(* Logix 5000 project; controller Receptivo vendor 1 type 14 code 106 rev 30.11; software revision 30.00; part 4 of 10 *)
(* tags used below, declared in another part *)
   Bit_Medianoche : BOOL;
   bit_ptobar : BOOL;
   Calendario : Hora_y_Fecha;
   Cola_Densidad_Bidon_Ayer : REAL[50];
   Cola_Densidad_Bidon_Fecha_Ayer : Hora_y_Fecha[50];
   Cola_Densidad_Bidones : REAL[50];
   Cola_Densidad_Bidones_Fecha : Hora_y_Fecha[50];
   Cola_Densidad_Elmar : REAL[50];
   Cola_Densidad_Elmar_Ayer : REAL[50];
   Cola_Densidad_Elmar_Fecha : Hora_y_Fecha[50];
   Cola_Densidad_Elmar_Fecha_Ayer : Hora_y_Fecha[50];
   Cola_Densidad_Fogg1 : REAL[50];
   Cola_Densidad_Fogg1_Ayer : REAL[50];
   Cola_Densidad_fogg1_Fecha : Hora_y_Fecha[50];
   Cola_Densidad_fogg1_Fecha_Ayer : Hora_y_Fecha[50];
   Cola_Densidad_Fogg2 : REAL[50];
   Cola_Densidad_Fogg2_Ayer : REAL[50];
   Cola_Densidad_fogg2_Fecha : Hora_y_Fecha[50];
   Cola_Densidad_fogg2_Fecha_Ayer : Hora_y_Fecha[50];
   Cola_Densidad_Karat : REAL[50];
   Cola_Densidad_Karat_Ayer : REAL[50];
   Cola_Densidad_Karat_Fecha : Hora_y_Fecha[50];
   Cola_Densidad_Karat_Fecha_Ayer : Hora_y_Fecha[50];
   Cola_Peso_Bidones : REAL[50];
   Cola_Peso_Caja_Bidon_Ayer : REAL[50];
   Cola_Peso_Caja_Elmar : REAL[50];
   Cola_Peso_Caja_Elmar_Ayer : REAL[50];
   Cola_Peso_Caja_Fogg1 : REAL[50];
   Cola_Peso_Caja_Fogg1_Ayer : REAL[50];
   Cola_Peso_Caja_Fogg2 : REAL[50];
   Cola_Peso_Caja_Fogg2_Ayer : REAL[50];
   Cola_Peso_Caja_Karat : REAL[50];
   Cola_Peso_Caja_Karat_Ayer : REAL[50];
   Cola_QAD_Densidad_Bidon_Ayer : STRING[50];
   Cola_QAD_Densidad_Bidones : STRING[50];
   Cola_QAD_Densidad_Elmar : STRING[50];
   Cola_QAD_Densidad_Elmar_Ayer : STRING[50];
   Cola_QAD_Densidad_Fogg1 : STRING[50];
   Cola_QAD_Densidad_Fogg1_Ayer : STRING[50];
   Cola_QAD_Densidad_Fogg2 : STRING[50];
   Cola_QAD_Densidad_Fogg2_Ayer : STRING[50];
   Cola_QAD_Densidad_Karat : STRING[50];
   Cola_QAD_Densidad_Karat_Ayer : STRING[50];
   Control_Densidad_Bidones : CONTROL;
   Control_Densidad_Elmar : CONTROL;
   Control_Densidad_Fogg1 : CONTROL;
   Control_Densidad_Fogg2 : CONTROL;
   Control_Densidad_Karat : CONTROL;
   Densidad_Bidon_1 : REAL;
   Densidad_Bidones : REAL;
   Densidad_Elmar : REAL;
   Densidad_Elmar_1 : REAL;
   Densidad_Elmar_OK : BOOL;
   Densidad_Fogg1 : REAL;
   Densidad_Fogg1_1 : REAL;
   Densidad_Fogg1_OK : BOOL;
   Densidad_Fogg2 : REAL;
   Densidad_Fogg2_1 : REAL;
   Densidad_Fogg2_OK : BOOL;
   Densidad_Karat : REAL;
   Densidad_Karat_1 : REAL;
   Densidad_Karat_OK : BOOL;
   Hora_Ingreso_Datos_Elmar : Hora_y_Fecha;
   Index_Bidones_Videojet : DINT;
   Index_Elmar_Videojet : DINT;
   Index_Fogg1_Videojet : DINT;
   Index_Fogg2_Videojet : DINT;
   Index_Karat_Videojet : DINT;
   Index_Karat_Videojet_Antiguo : DINT;
   Lote : DINT;
   Nuevo_Lote_Fogg1 : BOOL;
   ons_datos_mal_Bidones : BOOL;
   ons_datos_mal_elmar : BOOL;
   ons_datos_mal_Fogg1 : BOOL;
   ons_datos_mal_Fogg2 : BOOL;
   Ons_Datos_Mal_Karat : BOOL;
   ons_densidad_Fogg_1 : BOOL;
   Ons_Nuevo_Karat_Videojet : BOOL;
   Pesaje_Elmar_OK : BOOL;
   Pesaje_Fogg1_OK : BOOL;
   Pesaje_Fogg2_OK : BOOL;
   Pesaje_Karat_OK : BOOL;
   Peso_Bidones : REAL;
   Peso_Bidones_1 : REAL;
   Peso_Caja_Elmar : REAL;
   Peso_Caja_Elmar_1 : REAL;
   Peso_Caja_Fogg1 : REAL;
   Peso_Caja_Fogg1_1 : REAL;
   Peso_Caja_Fogg2 : REAL;
   Peso_Caja_Fogg2_1 : REAL;
   Peso_Caja_Karat : REAL;
   Peso_Caja_Karat_1 : REAL;
   Producido_Bidones_Ahora : UDT_Maestro;
   Producido_Elmar_Ahora : UDT_Maestro;
   Producido_Fogg1_Ahora : UDT_Maestro;
   Producido_Fogg2_Ahora : UDT_Maestro;
   Producido_Karat_Ahora : UDT_Maestro;
   Productos : UDT_Maestro[300];
   PV_Datos_Mal_Bidones : BOOL;
   PV_Datos_Mal_Elmar : BOOL;
   PV_Datos_Mal_Fogg1 : BOOL;
   PV_Datos_Mal_Fogg2 : BOOL;
   PV_Datos_Mal_Karat : BOOL;
   PV_Datos_Malos_Elmar : BOOL;
   PV_Datos_Malos_Fogg2 : BOOL;
   PV_Datos_Malos_Karat : BOOL;
   PV_Datos_Pesaje_Bidones : BOOL;
   PV_Datos_Pesaje_Elmar : BOOL;
   PV_Datos_Pesaje_Fogg1 : BOOL;
   PV_Datos_Pesaje_Fogg2 : BOOL;
   PV_Datos_Pesaje_Karat : BOOL;
   Slash : STRING;
   Timer_Datos_Bidones : TIMER;
   U_Fecha_Bidones : Hora_y_Fecha;
   U_Fecha_Elmar : Hora_y_Fecha;
   U_Fecha_Fogg1 : Hora_y_Fecha;
   U_Fecha_Fogg2 : Hora_y_Fecha;
   U_Fecha_Karat : Hora_y_Fecha;
   Un_Espacio : STRING;

PROGRAM Calculo_Produccion   (* main routine Principal_Calculo *)
VAR
   Entro_Datos_Pesaje_Bidones : BOOL;
   Entro_Datos_Pesaje_Elmar : BOOL;
   Entro_Datos_Pesaje_Fogg1 : BOOL;
   Entro_Datos_Pesaje_Fogg2 : BOOL;
   Entro_Datos_Pesaje_Karat : BOOL;
   Fecha_Cero : Hora_y_Fecha;
   Index_Bidones_Videojet_Antiguo : DINT;
   Index_Elmar_Videojet_Antiguo : DINT := 112;
   Index_Fogg1_Videojet_Antiguo : DINT := 203;
   Index_Fogg2_Videojet_Antiguo : DINT := 23;
   Nuevo_Lote_Bidones : BOOL;
   Nuevo_Lote_Elmar : BOOL;
   Nuevo_Lote_Fogg2 : BOOL;
   Nuevo_Lote_Karat : BOOL;
   ons_datos_elmar_malos : BOOL;
   ons_datos_fogg1_malos : BOOL;
   ons_datos_fogg2_malos : BOOL;
   Ons_Datos_Malos_Karat : BOOL;
   ons_densidad_bidones : BOOL;
   ons_densidad_elmar_1 : BOOL;
   ons_densidad_Fogg_2 : BOOL;
   Ons_Densidad_Karat : BOOL;
   ons_medianoche_Bidones : BOOL;
   ons_medianoche_Elmar : BOOL;
   ons_medianoche_Fogg1 : BOOL;
   ons_medianoche_Fogg2 : BOOL;
   Ons_Medianoche_Karat : BOOL;
   ons_nuevo_bidones_videojet : BOOL;
   ons_nuevo_elmar_videojet : BOOL;
   ons_nuevo_fogg1_videojet : BOOL;
   ons_nuevo_fogg2_videojet : BOOL;
   ons_peso_caja_elmar_1 : BOOL;
   Peso_Caja_Elmar_Entro : BOOL;
   PV_Datos_Malos_Fogg1 : BOOL;
   Salida_cola_densidad_elmar : REAL;
   Salida_peso_caja_elmar : REAL;
   Timer_Datos_1 : TIMER := (PRE := 600000);
   Timer_Datos_Fogg1 : TIMER := (PRE := 600000);
   Timer_Datos_Fogg2 : TIMER := (PRE := 600000);
   Timer_Datos_Karat : TIMER := (PRE := 600000);
END_VAR

ROUTINE Calculo_Pesaje_Bidones   (* ladder *)
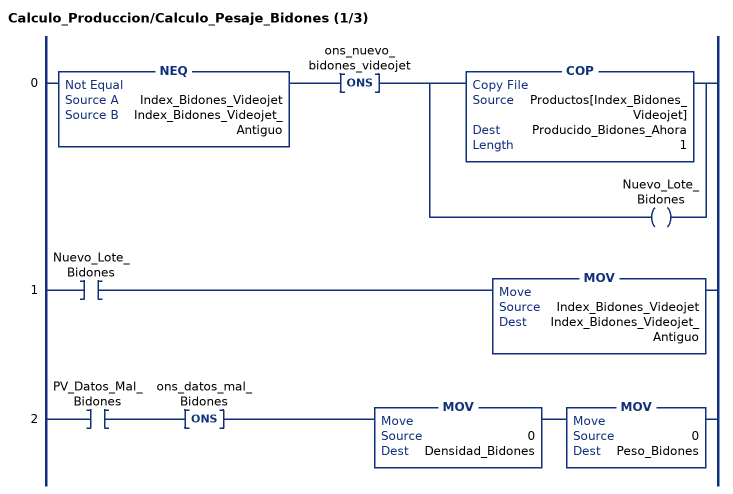
   0: NEQ(Index_Bidones_Videojet,Index_Bidones_Videojet_Antiguo)ONS(ons_nuevo_bidones_videojet)[COP(Productos[Index_Bidones_Videojet],Producido_Bidones_Ahora,1) ,OTE(Nuevo_Lote_Bidones) ];
   1: XIC(Nuevo_Lote_Bidones)MOV(Index_Bidones_Videojet,Index_Bidones_Videojet_Antiguo);
   2: XIC(PV_Datos_Mal_Bidones)ONS(ons_datos_mal_Bidones)MOV(0,Densidad_Bidones)MOV(0,Peso_Bidones);
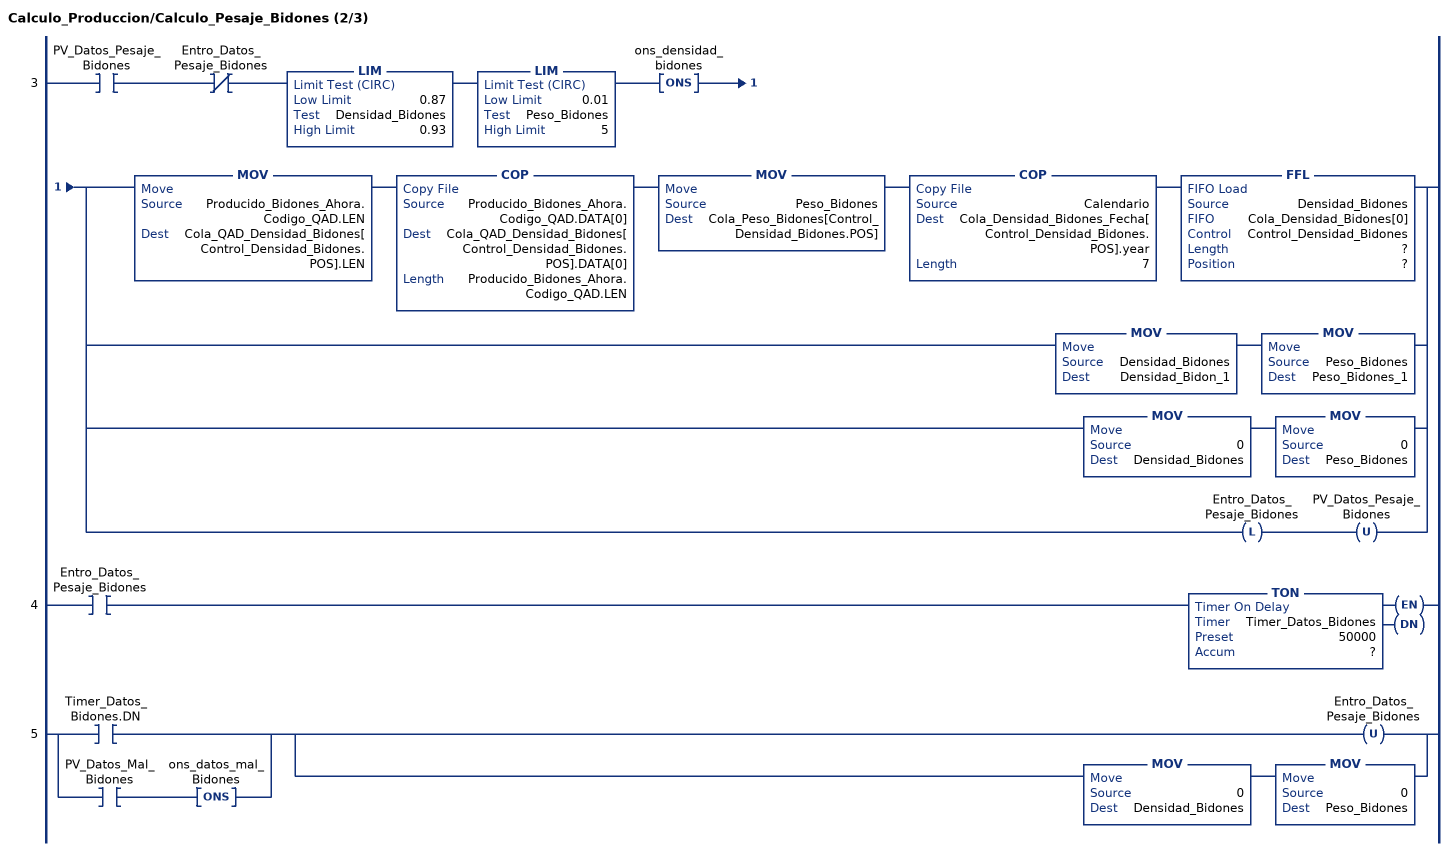
   3: XIC(PV_Datos_Pesaje_Bidones)XIO(Entro_Datos_Pesaje_Bidones)LIM(0.87,Densidad_Bidones,0.93)LIM(0.01,Peso_Bidones,5)ONS(ons_densidad_bidones)[MOV(Producido_Bidones_Ahora.Codigo_QAD.LEN,Cola_QAD_Densidad_Bidones[Control_Densidad_Bidones.POS].LEN) COP(Producido_Bidones_Ahora.Codigo_QAD.DATA[0],Cola_QAD_Densidad_Bidones[Control_Densidad_Bidones.POS].DATA[0],Producido_Bidones_Ahora.Codigo_QAD.LEN) MOV(Peso_Bidones,Cola_Peso_Bidones[Control_Densidad_Bidones.POS]) COP(Calendario,Cola_Densidad_Bidones_Fecha[Control_Densidad_Bidones.POS].year,7) FFL(Densidad_Bidones,Cola_Densidad_Bidones[0],Control_Densidad_Bidones,?,?) ,MOV(Densidad_Bidones,Densidad_Bidon_1) MOV(Peso_Bidones,Peso_Bidones_1) ,MOV(0,Densidad_Bidones) MOV(0,Peso_Bidones) ,OTL(Entro_Datos_Pesaje_Bidones) OTU(PV_Datos_Pesaje_Bidones) ];
   4: XIC(Entro_Datos_Pesaje_Bidones)TON(Timer_Datos_Bidones,?,?);
   5: [XIC(Timer_Datos_Bidones.DN) ,XIC(PV_Datos_Mal_Bidones) ONS(ons_datos_mal_Bidones) ][OTU(Entro_Datos_Pesaje_Bidones) ,MOV(0,Densidad_Bidones) MOV(0,Peso_Bidones) ];
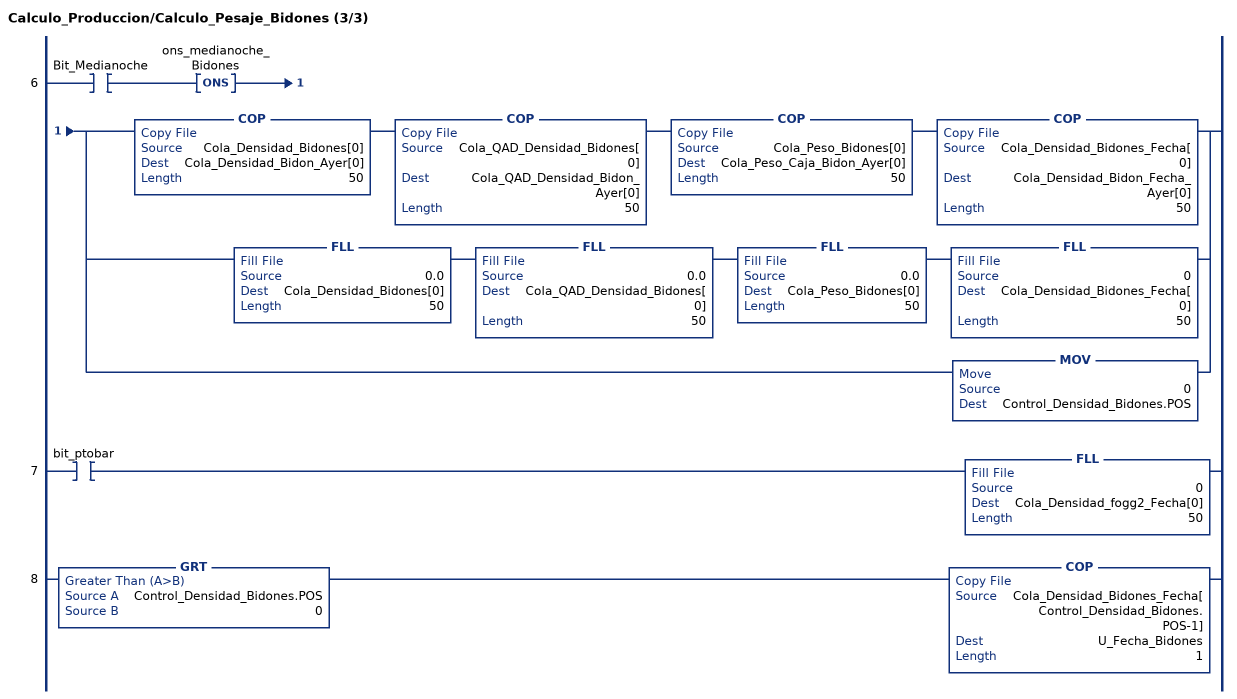
   6: XIC(Bit_Medianoche)ONS(ons_medianoche_Bidones)[COP(Cola_Densidad_Bidones[0],Cola_Densidad_Bidon_Ayer[0],50) COP(Cola_QAD_Densidad_Bidones[0],Cola_QAD_Densidad_Bidon_Ayer[0],50) COP(Cola_Peso_Bidones[0],Cola_Peso_Caja_Bidon_Ayer[0],50) COP(Cola_Densidad_Bidones_Fecha[0],Cola_Densidad_Bidon_Fecha_Ayer[0],50) ,FLL(0.0,Cola_Densidad_Bidones[0],50) FLL(0.0,Cola_QAD_Densidad_Bidones[0],50) FLL(0.0,Cola_Peso_Bidones[0],50) FLL(0,Cola_Densidad_Bidones_Fecha[0],50) ,MOV(0,Control_Densidad_Bidones.POS) ];
   7: XIC(bit_ptobar)FLL(0,Cola_Densidad_fogg2_Fecha[0],50);
   8: GRT(Control_Densidad_Bidones.POS,0)COP(Cola_Densidad_Bidones_Fecha[Control_Densidad_Bidones.POS-1],U_Fecha_Bidones,1);
END_ROUTINE

ROUTINE Calculo_Pesaje_Elmar   (* ladder *)
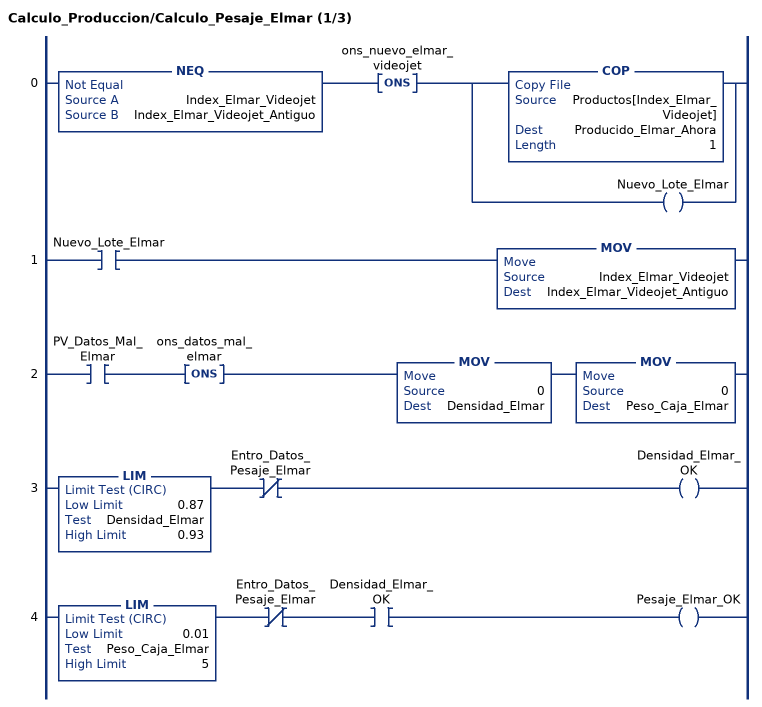
   0: NEQ(Index_Elmar_Videojet,Index_Elmar_Videojet_Antiguo)ONS(ons_nuevo_elmar_videojet)[COP(Productos[Index_Elmar_Videojet],Producido_Elmar_Ahora,1) ,OTE(Nuevo_Lote_Elmar) ];
   1: XIC(Nuevo_Lote_Elmar)MOV(Index_Elmar_Videojet,Index_Elmar_Videojet_Antiguo);
   2: XIC(PV_Datos_Mal_Elmar)ONS(ons_datos_mal_elmar)MOV(0,Densidad_Elmar)MOV(0,Peso_Caja_Elmar);
   3: LIM(0.87,Densidad_Elmar,0.93)XIO(Entro_Datos_Pesaje_Elmar)OTE(Densidad_Elmar_OK);
   4: LIM(0.01,Peso_Caja_Elmar,5)XIO(Entro_Datos_Pesaje_Elmar)XIC(Densidad_Elmar_OK)OTE(Pesaje_Elmar_OK);
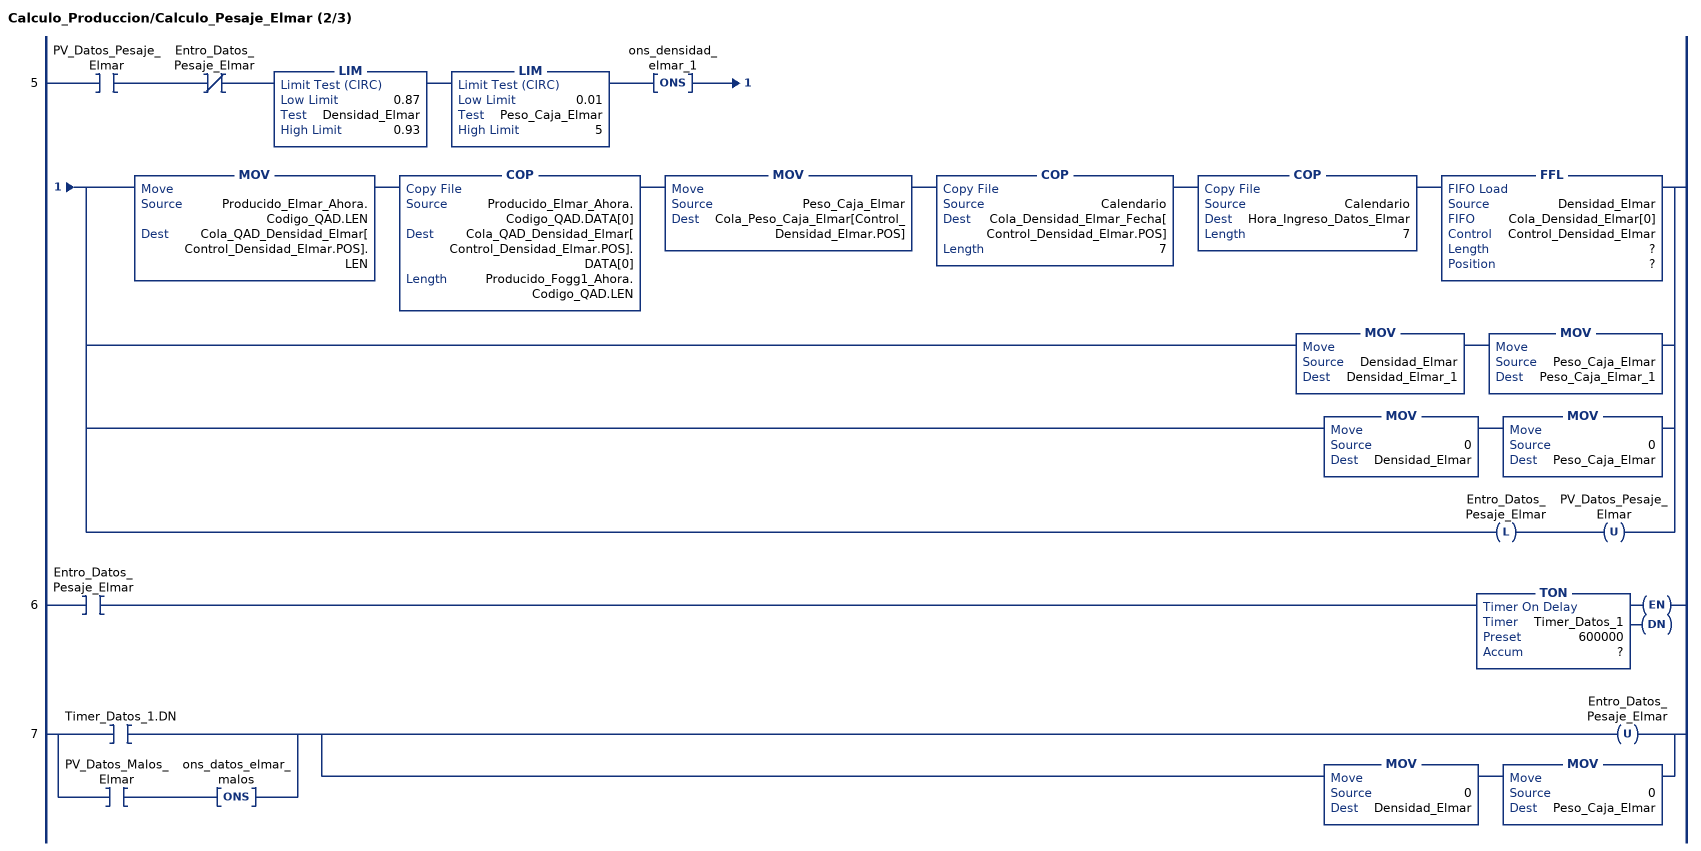
   5: XIC(PV_Datos_Pesaje_Elmar)XIO(Entro_Datos_Pesaje_Elmar)LIM(0.87,Densidad_Elmar,0.93)LIM(0.01,Peso_Caja_Elmar,5)ONS(ons_densidad_elmar_1)[MOV(Producido_Elmar_Ahora.Codigo_QAD.LEN,Cola_QAD_Densidad_Elmar[Control_Densidad_Elmar.POS].LEN) COP(Producido_Elmar_Ahora.Codigo_QAD.DATA[0],Cola_QAD_Densidad_Elmar[Control_Densidad_Elmar.POS].DATA[0],Producido_Fogg1_Ahora.Codigo_QAD.LEN) MOV(Peso_Caja_Elmar,Cola_Peso_Caja_Elmar[Control_Densidad_Elmar.POS]) COP(Calendario,Cola_Densidad_Elmar_Fecha[Control_Densidad_Elmar.POS],7) COP(Calendario,Hora_Ingreso_Datos_Elmar,7) FFL(Densidad_Elmar,Cola_Densidad_Elmar[0],Control_Densidad_Elmar,?,?) ,MOV(Densidad_Elmar,Densidad_Elmar_1) MOV(Peso_Caja_Elmar,Peso_Caja_Elmar_1) ,MOV(0,Densidad_Elmar) MOV(0,Peso_Caja_Elmar) ,OTL(Entro_Datos_Pesaje_Elmar) OTU(PV_Datos_Pesaje_Elmar) ];
   6: XIC(Entro_Datos_Pesaje_Elmar)TON(Timer_Datos_1,?,?);
   7: [XIC(Timer_Datos_1.DN) ,XIC(PV_Datos_Malos_Elmar) ONS(ons_datos_elmar_malos) ][OTU(Entro_Datos_Pesaje_Elmar) ,MOV(0,Densidad_Elmar) MOV(0,Peso_Caja_Elmar) ];
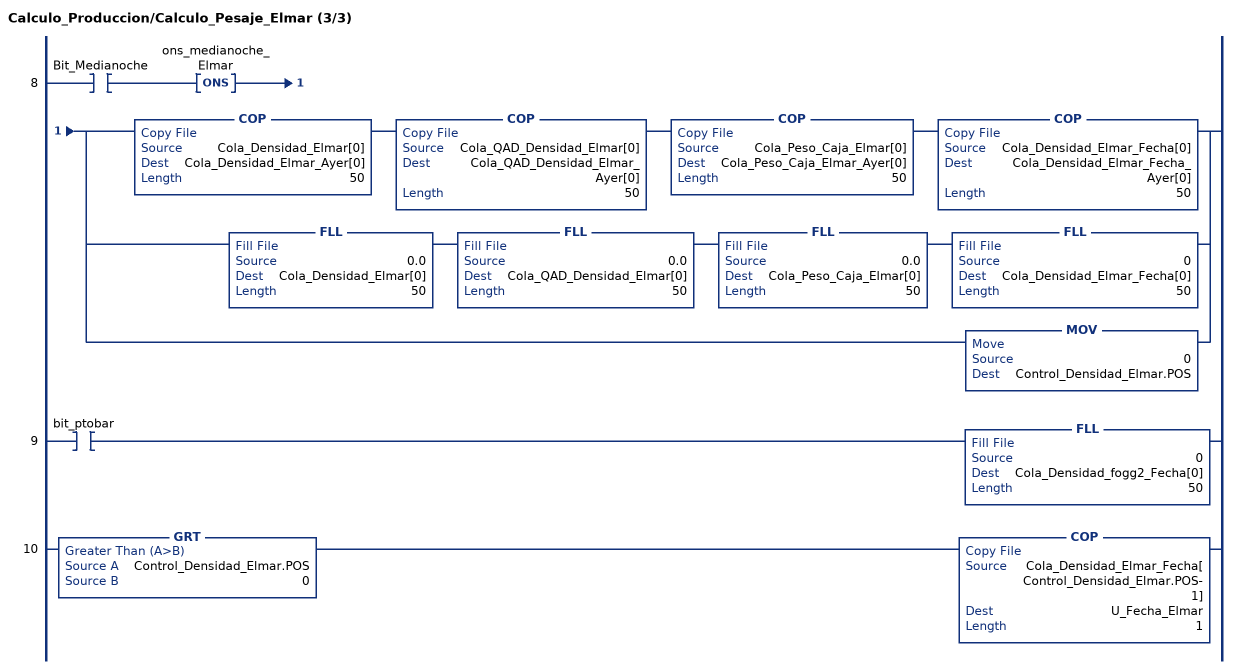
   8: XIC(Bit_Medianoche)ONS(ons_medianoche_Elmar)[COP(Cola_Densidad_Elmar[0],Cola_Densidad_Elmar_Ayer[0],50) COP(Cola_QAD_Densidad_Elmar[0],Cola_QAD_Densidad_Elmar_Ayer[0],50) COP(Cola_Peso_Caja_Elmar[0],Cola_Peso_Caja_Elmar_Ayer[0],50) COP(Cola_Densidad_Elmar_Fecha[0],Cola_Densidad_Elmar_Fecha_Ayer[0],50) ,FLL(0.0,Cola_Densidad_Elmar[0],50) FLL(0.0,Cola_QAD_Densidad_Elmar[0],50) FLL(0.0,Cola_Peso_Caja_Elmar[0],50) FLL(0,Cola_Densidad_Elmar_Fecha[0],50) ,MOV(0,Control_Densidad_Elmar.POS) ];
   9: XIC(bit_ptobar)FLL(0,Cola_Densidad_fogg2_Fecha[0],50);
   10: GRT(Control_Densidad_Elmar.POS,0)COP(Cola_Densidad_Elmar_Fecha[Control_Densidad_Elmar.POS-1],U_Fecha_Elmar,1);
END_ROUTINE

ROUTINE Calculo_Pesaje_Fogg1   (* ladder *)
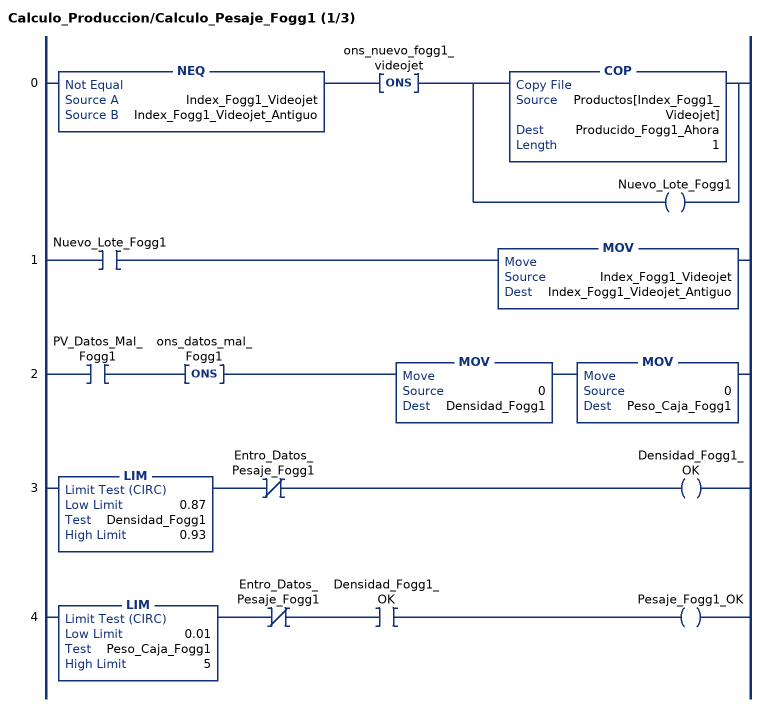
   0: NEQ(Index_Fogg1_Videojet,Index_Fogg1_Videojet_Antiguo)ONS(ons_nuevo_fogg1_videojet)[COP(Productos[Index_Fogg1_Videojet],Producido_Fogg1_Ahora,1) ,OTE(Nuevo_Lote_Fogg1) ];
   1: XIC(Nuevo_Lote_Fogg1)MOV(Index_Fogg1_Videojet,Index_Fogg1_Videojet_Antiguo);
   2: XIC(PV_Datos_Mal_Fogg1)ONS(ons_datos_mal_Fogg1)MOV(0,Densidad_Fogg1)MOV(0,Peso_Caja_Fogg1);
   3: LIM(0.87,Densidad_Fogg1,0.93)XIO(Entro_Datos_Pesaje_Fogg1)OTE(Densidad_Fogg1_OK);
   4: LIM(0.01,Peso_Caja_Fogg1,5)XIO(Entro_Datos_Pesaje_Fogg1)XIC(Densidad_Fogg1_OK)OTE(Pesaje_Fogg1_OK);
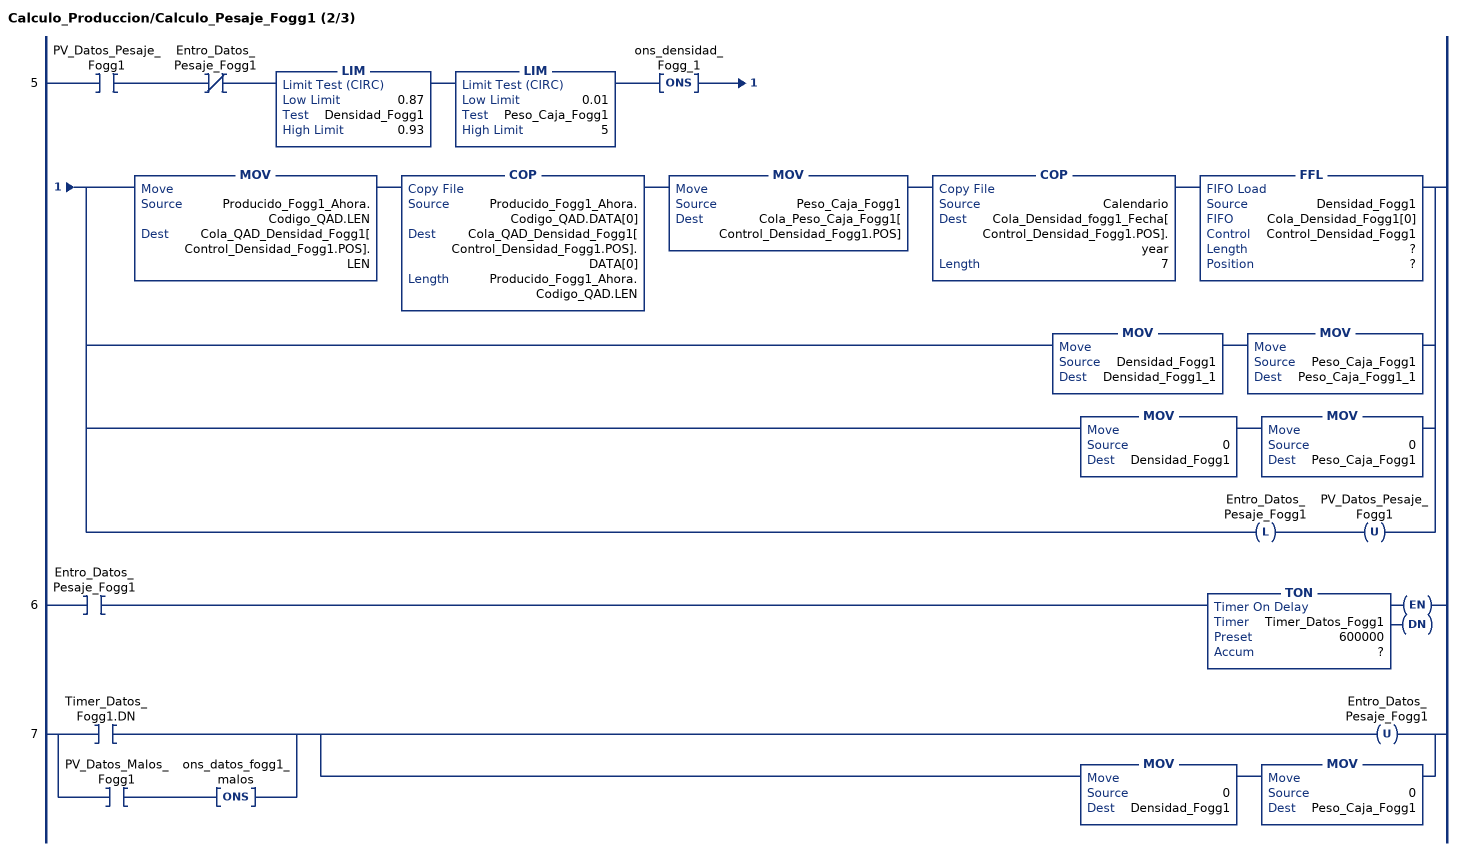
   5: XIC(PV_Datos_Pesaje_Fogg1)XIO(Entro_Datos_Pesaje_Fogg1)LIM(0.87,Densidad_Fogg1,0.93)LIM(0.01,Peso_Caja_Fogg1,5)ONS(ons_densidad_Fogg_1)[MOV(Producido_Fogg1_Ahora.Codigo_QAD.LEN,Cola_QAD_Densidad_Fogg1[Control_Densidad_Fogg1.POS].LEN) COP(Producido_Fogg1_Ahora.Codigo_QAD.DATA[0],Cola_QAD_Densidad_Fogg1[Control_Densidad_Fogg1.POS].DATA[0],Producido_Fogg1_Ahora.Codigo_QAD.LEN) MOV(Peso_Caja_Fogg1,Cola_Peso_Caja_Fogg1[Control_Densidad_Fogg1.POS]) COP(Calendario,Cola_Densidad_fogg1_Fecha[Control_Densidad_Fogg1.POS].year,7) FFL(Densidad_Fogg1,Cola_Densidad_Fogg1[0],Control_Densidad_Fogg1,?,?) ,MOV(Densidad_Fogg1,Densidad_Fogg1_1) MOV(Peso_Caja_Fogg1,Peso_Caja_Fogg1_1) ,MOV(0,Densidad_Fogg1) MOV(0,Peso_Caja_Fogg1) ,OTL(Entro_Datos_Pesaje_Fogg1) OTU(PV_Datos_Pesaje_Fogg1) ];
   6: XIC(Entro_Datos_Pesaje_Fogg1)TON(Timer_Datos_Fogg1,?,?);
   7: [XIC(Timer_Datos_Fogg1.DN) ,XIC(PV_Datos_Malos_Fogg1) ONS(ons_datos_fogg1_malos) ][OTU(Entro_Datos_Pesaje_Fogg1) ,MOV(0,Densidad_Fogg1) MOV(0,Peso_Caja_Fogg1) ];
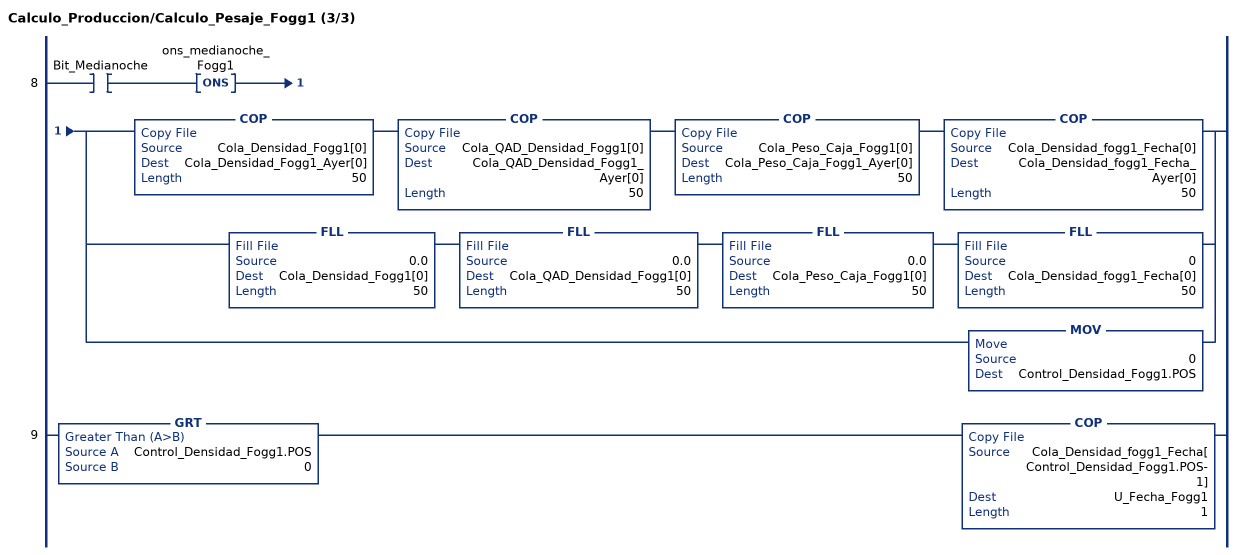
   8: XIC(Bit_Medianoche)ONS(ons_medianoche_Fogg1)[COP(Cola_Densidad_Fogg1[0],Cola_Densidad_Fogg1_Ayer[0],50) COP(Cola_QAD_Densidad_Fogg1[0],Cola_QAD_Densidad_Fogg1_Ayer[0],50) COP(Cola_Peso_Caja_Fogg1[0],Cola_Peso_Caja_Fogg1_Ayer[0],50) COP(Cola_Densidad_fogg1_Fecha[0],Cola_Densidad_fogg1_Fecha_Ayer[0],50) ,FLL(0.0,Cola_Densidad_Fogg1[0],50) FLL(0.0,Cola_QAD_Densidad_Fogg1[0],50) FLL(0.0,Cola_Peso_Caja_Fogg1[0],50) FLL(0,Cola_Densidad_fogg1_Fecha[0],50) ,MOV(0,Control_Densidad_Fogg1.POS) ];
   9: GRT(Control_Densidad_Fogg1.POS,0)COP(Cola_Densidad_fogg1_Fecha[Control_Densidad_Fogg1.POS-1],U_Fecha_Fogg1,1);
END_ROUTINE

ROUTINE Calculo_Pesaje_Fogg2   (* ladder *)
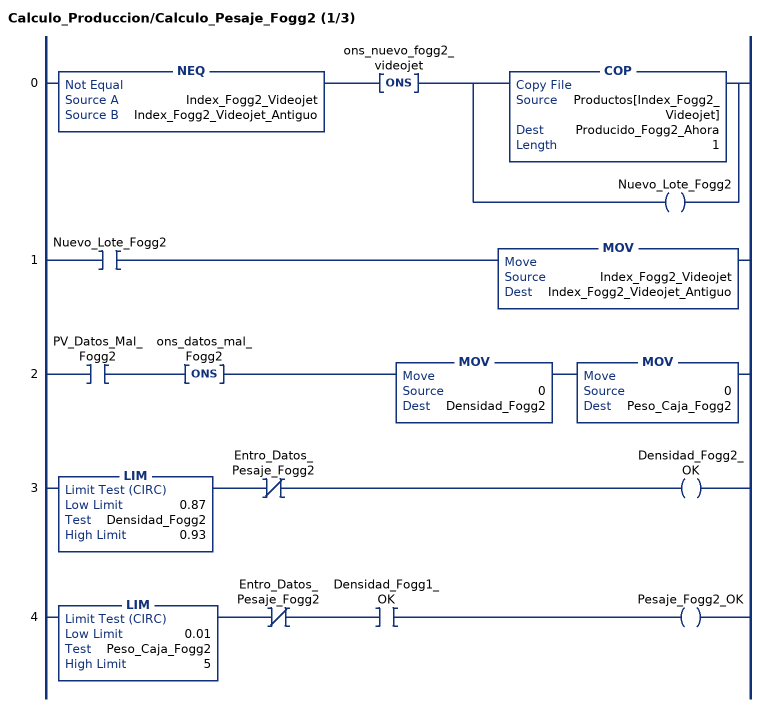
   0: NEQ(Index_Fogg2_Videojet,Index_Fogg2_Videojet_Antiguo)ONS(ons_nuevo_fogg2_videojet)[COP(Productos[Index_Fogg2_Videojet],Producido_Fogg2_Ahora,1) ,OTE(Nuevo_Lote_Fogg2) ];
   1: XIC(Nuevo_Lote_Fogg2)MOV(Index_Fogg2_Videojet,Index_Fogg2_Videojet_Antiguo);
   2: XIC(PV_Datos_Mal_Fogg2)ONS(ons_datos_mal_Fogg2)MOV(0,Densidad_Fogg2)MOV(0,Peso_Caja_Fogg2);
   3: LIM(0.87,Densidad_Fogg2,0.93)XIO(Entro_Datos_Pesaje_Fogg2)OTE(Densidad_Fogg2_OK);
   4: LIM(0.01,Peso_Caja_Fogg2,5)XIO(Entro_Datos_Pesaje_Fogg2)XIC(Densidad_Fogg1_OK)OTE(Pesaje_Fogg2_OK);
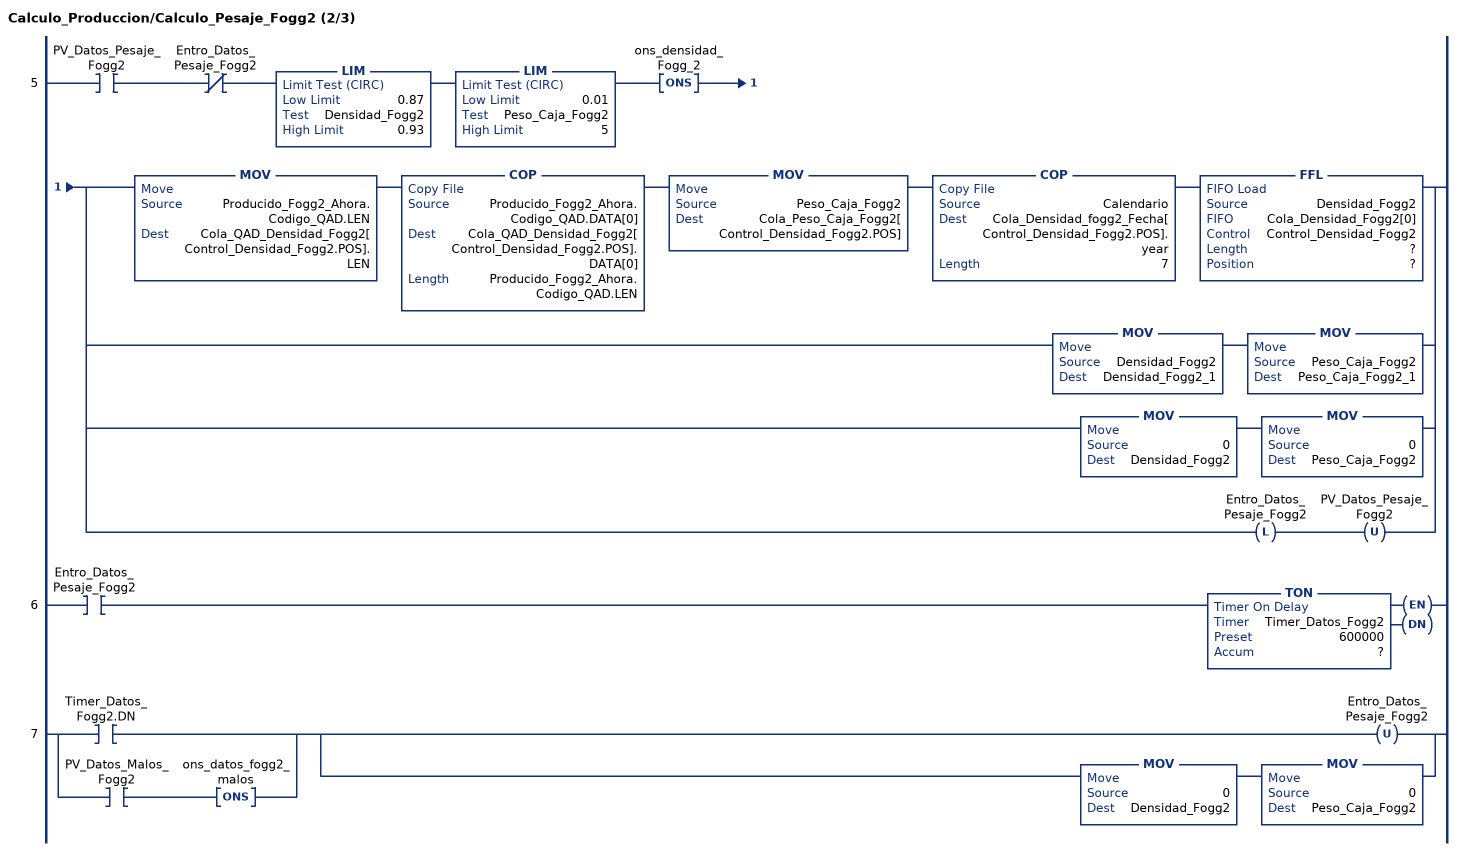
   5: XIC(PV_Datos_Pesaje_Fogg2)XIO(Entro_Datos_Pesaje_Fogg2)LIM(0.87,Densidad_Fogg2,0.93)LIM(0.01,Peso_Caja_Fogg2,5)ONS(ons_densidad_Fogg_2)[MOV(Producido_Fogg2_Ahora.Codigo_QAD.LEN,Cola_QAD_Densidad_Fogg2[Control_Densidad_Fogg2.POS].LEN) COP(Producido_Fogg2_Ahora.Codigo_QAD.DATA[0],Cola_QAD_Densidad_Fogg2[Control_Densidad_Fogg2.POS].DATA[0],Producido_Fogg2_Ahora.Codigo_QAD.LEN) MOV(Peso_Caja_Fogg2,Cola_Peso_Caja_Fogg2[Control_Densidad_Fogg2.POS]) COP(Calendario,Cola_Densidad_fogg2_Fecha[Control_Densidad_Fogg2.POS].year,7) FFL(Densidad_Fogg2,Cola_Densidad_Fogg2[0],Control_Densidad_Fogg2,?,?) ,MOV(Densidad_Fogg2,Densidad_Fogg2_1) MOV(Peso_Caja_Fogg2,Peso_Caja_Fogg2_1) ,MOV(0,Densidad_Fogg2) MOV(0,Peso_Caja_Fogg2) ,OTL(Entro_Datos_Pesaje_Fogg2) OTU(PV_Datos_Pesaje_Fogg2) ];
   6: XIC(Entro_Datos_Pesaje_Fogg2)TON(Timer_Datos_Fogg2,?,?);
   7: [XIC(Timer_Datos_Fogg2.DN) ,XIC(PV_Datos_Malos_Fogg2) ONS(ons_datos_fogg2_malos) ][OTU(Entro_Datos_Pesaje_Fogg2) ,MOV(0,Densidad_Fogg2) MOV(0,Peso_Caja_Fogg2) ];
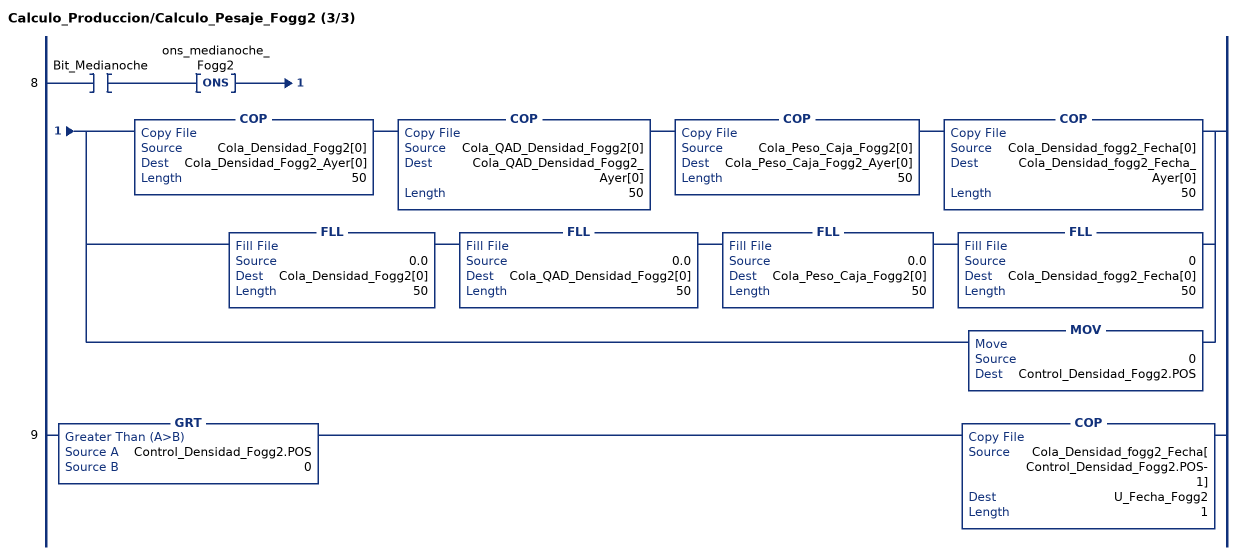
   8: XIC(Bit_Medianoche)ONS(ons_medianoche_Fogg2)[COP(Cola_Densidad_Fogg2[0],Cola_Densidad_Fogg2_Ayer[0],50) COP(Cola_QAD_Densidad_Fogg2[0],Cola_QAD_Densidad_Fogg2_Ayer[0],50) COP(Cola_Peso_Caja_Fogg2[0],Cola_Peso_Caja_Fogg2_Ayer[0],50) COP(Cola_Densidad_fogg2_Fecha[0],Cola_Densidad_fogg2_Fecha_Ayer[0],50) ,FLL(0.0,Cola_Densidad_Fogg2[0],50) FLL(0.0,Cola_QAD_Densidad_Fogg2[0],50) FLL(0.0,Cola_Peso_Caja_Fogg2[0],50) FLL(0,Cola_Densidad_fogg2_Fecha[0],50) ,MOV(0,Control_Densidad_Fogg2.POS) ];
   9: GRT(Control_Densidad_Fogg2.POS,0)COP(Cola_Densidad_fogg2_Fecha[Control_Densidad_Fogg2.POS-1],U_Fecha_Fogg2,1);
END_ROUTINE

ROUTINE Calculo_Pesaje_Karat   (* ladder *)
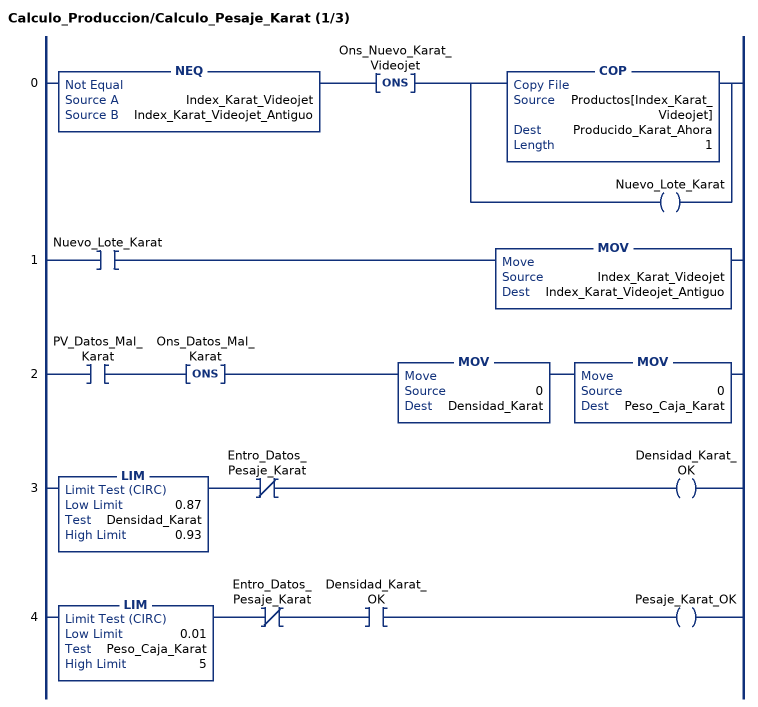
   0: NEQ(Index_Karat_Videojet,Index_Karat_Videojet_Antiguo)ONS(Ons_Nuevo_Karat_Videojet)[COP(Productos[Index_Karat_Videojet],Producido_Karat_Ahora,1) ,OTE(Nuevo_Lote_Karat) ];
   1: XIC(Nuevo_Lote_Karat)MOV(Index_Karat_Videojet,Index_Karat_Videojet_Antiguo);
   2: XIC(PV_Datos_Mal_Karat)ONS(Ons_Datos_Mal_Karat)MOV(0,Densidad_Karat)MOV(0,Peso_Caja_Karat);
   3: LIM(0.87,Densidad_Karat,0.93)XIO(Entro_Datos_Pesaje_Karat)OTE(Densidad_Karat_OK);
   4: LIM(0.01,Peso_Caja_Karat,5)XIO(Entro_Datos_Pesaje_Karat)XIC(Densidad_Karat_OK)OTE(Pesaje_Karat_OK);
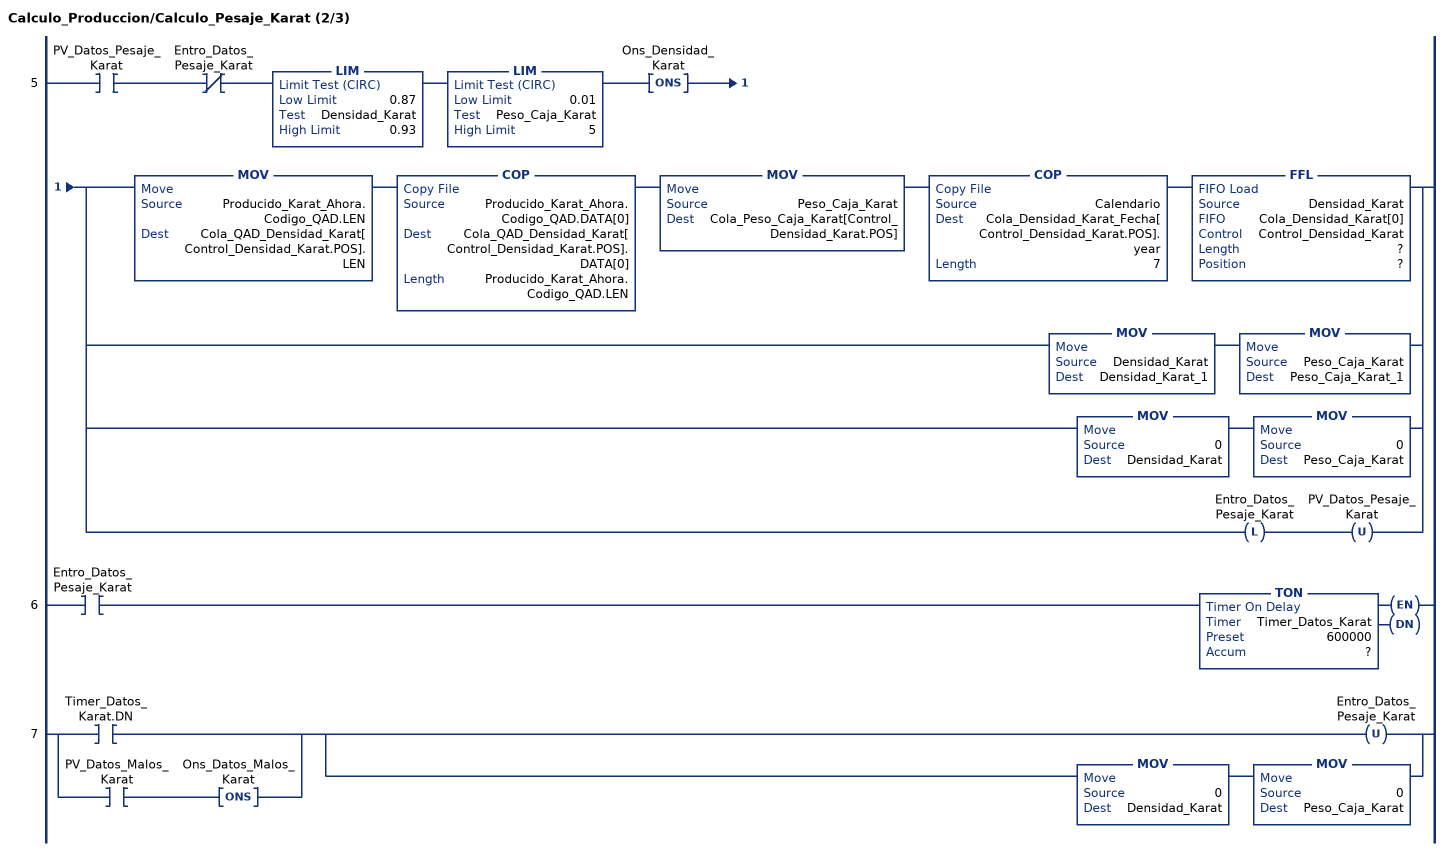
   5: XIC(PV_Datos_Pesaje_Karat)XIO(Entro_Datos_Pesaje_Karat)LIM(0.87,Densidad_Karat,0.93)LIM(0.01,Peso_Caja_Karat,5)ONS(Ons_Densidad_Karat)[MOV(Producido_Karat_Ahora.Codigo_QAD.LEN,Cola_QAD_Densidad_Karat[Control_Densidad_Karat.POS].LEN) COP(Producido_Karat_Ahora.Codigo_QAD.DATA[0],Cola_QAD_Densidad_Karat[Control_Densidad_Karat.POS].DATA[0],Producido_Karat_Ahora.Codigo_QAD.LEN) MOV(Peso_Caja_Karat,Cola_Peso_Caja_Karat[Control_Densidad_Karat.POS]) COP(Calendario,Cola_Densidad_Karat_Fecha[Control_Densidad_Karat.POS].year,7) FFL(Densidad_Karat,Cola_Densidad_Karat[0],Control_Densidad_Karat,?,?) ,MOV(Densidad_Karat,Densidad_Karat_1) MOV(Peso_Caja_Karat,Peso_Caja_Karat_1) ,MOV(0,Densidad_Karat) MOV(0,Peso_Caja_Karat) ,OTL(Entro_Datos_Pesaje_Karat) OTU(PV_Datos_Pesaje_Karat) ];
   6: XIC(Entro_Datos_Pesaje_Karat)TON(Timer_Datos_Karat,?,?);
   7: [XIC(Timer_Datos_Karat.DN) ,XIC(PV_Datos_Malos_Karat) ONS(Ons_Datos_Malos_Karat) ][OTU(Entro_Datos_Pesaje_Karat) ,MOV(0,Densidad_Karat) MOV(0,Peso_Caja_Karat) ];
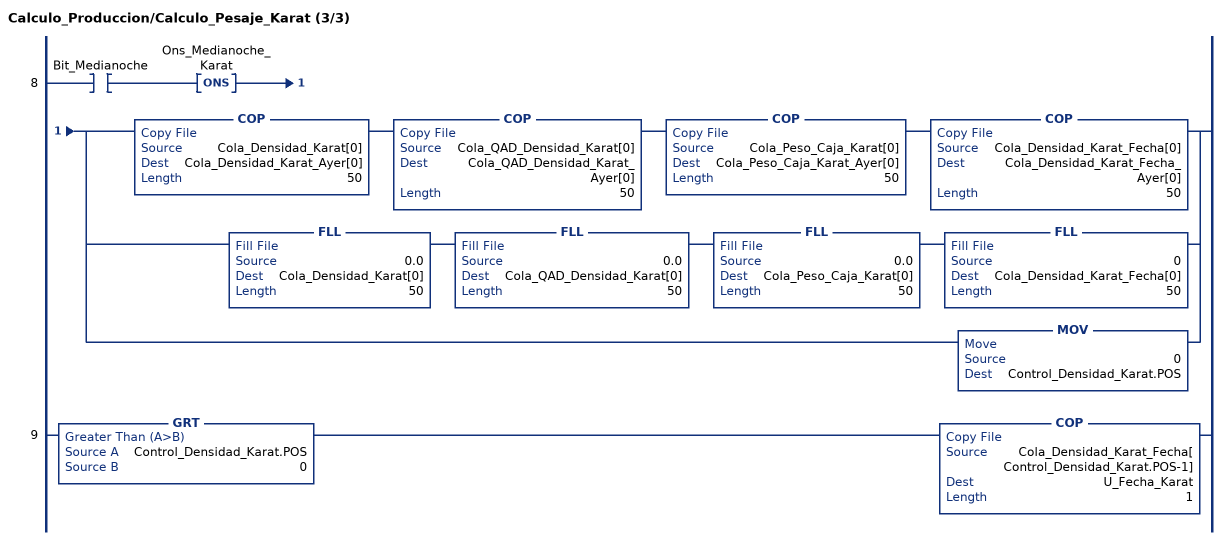
   8: XIC(Bit_Medianoche)ONS(Ons_Medianoche_Karat)[COP(Cola_Densidad_Karat[0],Cola_Densidad_Karat_Ayer[0],50) COP(Cola_QAD_Densidad_Karat[0],Cola_QAD_Densidad_Karat_Ayer[0],50) COP(Cola_Peso_Caja_Karat[0],Cola_Peso_Caja_Karat_Ayer[0],50) COP(Cola_Densidad_Karat_Fecha[0],Cola_Densidad_Karat_Fecha_Ayer[0],50) ,FLL(0.0,Cola_Densidad_Karat[0],50) FLL(0.0,Cola_QAD_Densidad_Karat[0],50) FLL(0.0,Cola_Peso_Caja_Karat[0],50) FLL(0,Cola_Densidad_Karat_Fecha[0],50) ,MOV(0,Control_Densidad_Karat.POS) ];
   9: GRT(Control_Densidad_Karat.POS,0)COP(Cola_Densidad_Karat_Fecha[Control_Densidad_Karat.POS-1],U_Fecha_Karat,1);
END_ROUTINE

ROUTINE Principal_Calculo   (* ladder *)
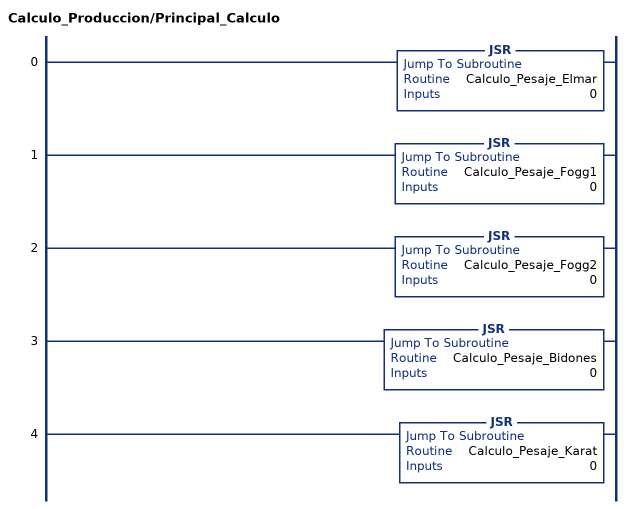
   0: JSR(Calculo_Pesaje_Elmar,0);
   1: JSR(Calculo_Pesaje_Fogg1,0);
   2: JSR(Calculo_Pesaje_Fogg2,0);
   3: JSR(Calculo_Pesaje_Bidones,0);
   4: JSR(Calculo_Pesaje_Karat,0);
END_ROUTINE
END_PROGRAM

PROGRAM MainProgram   (* main routine MainRoutine *)
VAR
   borrar : BOOL;
   Codigo_QAD1_Espacios : DINT := 112;
   Codigo_QAD3_Espacios : DINT := 112;
   Codigo_QAD4_Espacios : DINT := 112;
   Descripcion1_Espacios : DINT := 79;
   Descripcion2_Espacios : DINT := 73;
   Descripcion3_Espacios : DINT := 73;
   Descripcion4_Espacios : DINT := 66;
   dia_prueba : STRING := '01';
   End_Printing_2 : BOOL;
   Final_Print_1 : BOOL;
   Final_Print_2 : BOOL;
   Final_Print_3 : BOOL;
   Final_Print_4 : BOOL;
   Index_Print_1 : DINT;
   Index_Print_2 : DINT;
   Numero_Espacios_Descripcion_1 : DINT := 10;
   Numero_Espacios_Descripcion_2 : DINT := 16;
   Numero_Espacios_Descripcion_3 : DINT := 16;
   Numero_Espacios_Descripcion_4 : DINT := 23;
   Numero_Espacios_QAD1 : DINT;
   Numero_Espacios_QAD2 : DINT;
   Numero_Espacios_QAD3 : DINT;
   Numero_Espacios_QAD4 : DINT;
   Ons_Cola1 : BOOL;
   ons_imprimiendo : BOOL;
   ons_nuevo_dia : BOOL;
   ons_print1 : BOOL;
   ons_print1_aux : BOOL;
   ons_print2 : BOOL;
   ons_print2_2 : BOOL;
   ons_print2_aux : BOOL;
   ons_print3 : BOOL;
   ons_print3_aux : BOOL;
   ons_print4 : BOOL;
   ons_print4_aux : BOOL;
   ons_start_printing2 : BOOL;
   Print1_Ejecute : BOOL;
   Print1_OK : BOOL;
   Print2_Ejecute : BOOL;
   Print2_OK : BOOL;
   Print3_Ejecute : BOOL;
   Print3_OK : BOOL;
   Print4_Ejecute : BOOL;
   Print4_OK : BOOL;
   Printing2 : BOOL;
   Printing_1 : BOOL;
   Printing_2 : BOOL;
   Printing_3 : BOOL;
   Printing_4 : BOOL;
   Salida_Cola_Est_1 : UDT_COLA := (Fecha.year := 2019, Fecha.Mes := 1, Fecha.Dia := 5, Fecha.Hora := 12, Fecha.Minuto := 21, Fecha.Segundo := 50, Fecha.Milisegundos := 123163, Lote := 5, Operador := 5, Descripcion := 'La Muneca Caja 6 x 3000 cm3 FF', EAN14 := '17702179009203', QAD := '10140', Peso_Real := 867.0, Peso_Teorico := 869.0, No_Cajas := 50, Clima := 2, Consec := 97);
   Salida_Cola_Est_2 : UDT_COLA := (Fecha.year := 2021, Fecha.Mes := 5, Fecha.Dia := 6, Fecha.Minuto := 42, Fecha.Segundo := 51, Fecha.Milisegundos := 839426, Lote := 126, Operador := 5, Descripcion := 'MiD$EDa 24 x 500 cm3', EAN14 := '17705946719384', QAD := '634210', Peso_Real := 35.0, Peso_Teorico := 35.0, No_Cajas := 3, Clima := 1, Consec := 6, Envase := 500, Envases_x_Caja := 24, Densidad_Medida := 0.9152, Linea := 1);
   Salida_Cola_Est_3 : UDT_COLA := (Fecha.year := 2021, Fecha.Mes := 5, Fecha.Dia := 7, Fecha.Hora := 6, Fecha.Minuto := 43, Fecha.Segundo := 12, Fecha.Milisegundos := 399243, Lote := 127, Operador := 5, Descripcion := 'Alegr$EDa Caja 6 x 3000 cm3  - Costa', EAN14 := '17702161043987', QAD := '600300', Peso_Real := 513.0, Peso_Teorico := 519.0, No_Cajas := 30, Consec := 54, Envase := 3000, Envases_x_Caja := 6, Densidad_Medida := 0.9152, Linea := 3);
   Salida_Cola_Est_4 : UDT_COLA := (Fecha.year := 2021, Fecha.Mes := 5, Fecha.Dia := 24, Fecha.Hora := 11, Fecha.Minuto := 32, Fecha.Segundo := 31, Fecha.Milisegundos := 461899, Lote := 144, Operador := 6, Descripcion := 'Aceite Vegetal Torino  Exp.', EAN14 := '17702161820113', QAD := '607020', Peso_Real := 790.0, Peso_Teorico := 786.0, No_Cajas := 48, Consec := 35, Envase := 17250, Envases_x_Caja := 1, Densidad_Medida := 0.9148, Linea := 5);
END_VAR

ROUTINE Charateres_Fijos   (* ladder *)
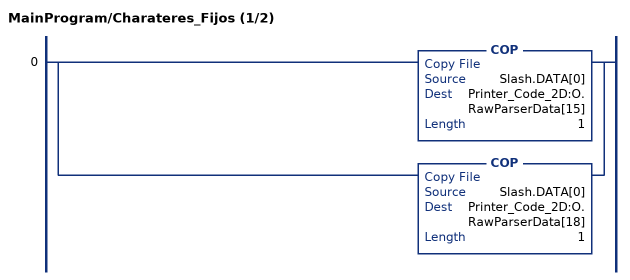
   0: [COP(Slash.DATA[0],Printer_Code_2D:O.RawParserData[15],1) ,COP(Slash.DATA[0],Printer_Code_2D:O.RawParserData[18],1) ];
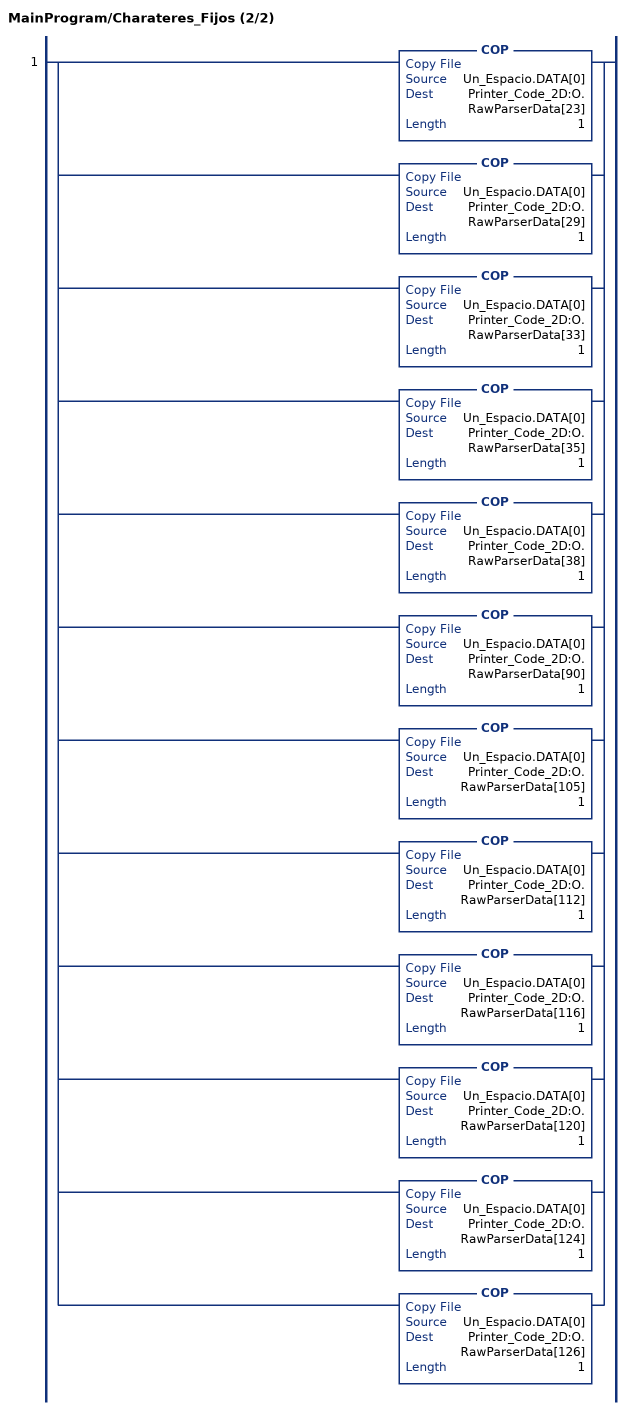
   1: [COP(Un_Espacio.DATA[0],Printer_Code_2D:O.RawParserData[23],1) ,COP(Un_Espacio.DATA[0],Printer_Code_2D:O.RawParserData[29],1) ,COP(Un_Espacio.DATA[0],Printer_Code_2D:O.RawParserData[33],1) ,COP(Un_Espacio.DATA[0],Printer_Code_2D:O.RawParserData[35],1) ,COP(Un_Espacio.DATA[0],Printer_Code_2D:O.RawParserData[38],1) ,COP(Un_Espacio.DATA[0],Printer_Code_2D:O.RawParserData[90],1) ,COP(Un_Espacio.DATA[0],Printer_Code_2D:O.RawParserData[105],1) ,COP(Un_Espacio.DATA[0],Printer_Code_2D:O.RawParserData[112],1) ,COP(Un_Espacio.DATA[0],Printer_Code_2D:O.RawParserData[116],1) ,COP(Un_Espacio.DATA[0],Printer_Code_2D:O.RawParserData[120],1) ,COP(Un_Espacio.DATA[0],Printer_Code_2D:O.RawParserData[124],1) ,COP(Un_Espacio.DATA[0],Printer_Code_2D:O.RawParserData[126],1) ];
END_ROUTINE
